(* IEC 61131-3 sources: Std_PalletMover/Class/CntrlAuxHmi, 1 file *)

(* ---- CntrlAuxHmi.st ---- *)
(*!
<Class
	Name               = "CntrlAuxHmi"
	Revision           = "0.0"
	RealtimeTask       = "false"
	CyclicTask         = "false"
	BackgroundTask     = "false"
	Sigmatek           = "false"
	OSInterface        = "false"
	HighPriority       = "false"
	Automatic          = "false"
	UpdateMode         = "Prescan"
	SharedCommandTable = "true"
	Objectsize         = "(960,120)">
	<Channels>
		<Server Name="AgvState" Visualized="false" Initialize="false" WriteProtected="true" Retentive="false"/>
		<Server Name="ErrorMessage" Visualized="false" Initialize="false" WriteProtected="true" Retentive="false"/>
		<Client Name="ToConfiguration" Required="true" Internal="false"/>
		<Client Name="ToMqttInterface" Required="true" Internal="false"/>
		<Client Name="ToSettings" Required="true" Internal="false"/>
	</Channels>
	<Network Name="CntrlAuxHmi">
		<!-- List of Components in this network -->
		<Components>
			<Object
				Name       = "_base"
				Class      = "AuxBase"
				Position   = "(218,120)"
				Visualized = "false">
				<Channels>
					<Server Name="ToObject"/>
					<Client Name="op_LogData"/>
					<Client Name="p_NextObject"/>
				</Channels>
			</Object>
		</Components>
		<Comments>
		</Comments>
		<!-- List of Connections in this network -->
		<Connections>
			<Connection Source="this.ToObject" Destination="_base.ToObject" Vertices="(976,210),(804,210),"/>
			<Connection Source="_base.op_LogData" Destination="this.op_LogData" Vertices="(218,210),(38,210),"/>
			<Connection Source="_base.p_NextObject" Destination="this.p_NextObject" Vertices="(218,270),(38,270),"/>
		</Connections>
		<!-- Headerfiles -->
		<Options>
		</Options>
	</Network>
</Class>
*)
#pragma using AuxBase

CntrlAuxHmi : CLASS
: AuxBase
  //Servers:
	ErrorMessage 	: SvrCh_DINT;
	AgvState 	: SvrCh_DINT;
  //Clients:
	ToConfiguration 	: CltChCmd_AgvConfig;
	ToSettings 	: CltChCmd_AgvSettings;
	ToMqttInterface 	: CltChCmd_MqttInterface;
  //Variables:
  //Functions:

	FUNCTION GetDataFromMqttchanel;
  //Tables:
	FUNCTION @STD
		VAR_OUTPUT
			ret_code	: CONFSTATES;
		END_VAR;
	FUNCTION GLOBAL TAB @CT_;
END_CLASS;

#pragma usingLtd AgvConfig
#pragma usingLtd AgvSettings
#pragma usingLtd MqttInterface

FUNCTION CntrlAuxHmi::GetDataFromMqttchanel

END_FUNCTION
